Yaskawa INFORM job: R1_W63-A2(130,-90)(JEDENR)KM-OK.JBI

/JOB
//NAME R1_W63-A2(130,-90)(JEDENR)KM-OK
///FOLDERNAME KRIS-SCIANA
//POS
///NPOS 116,116,0,5,0,0
///TOOL 0
///POSTYPE PULSE
///PULSE
C00000=-63639,-75448,-57109,45781,44405,52131
C00001=-94617,-44761,-17381,50840,21971,50320
C00002=-94032,-38268,-10140,52496,20938,49575
C00003=-93501,-34314,-6346,52601,20454,49570
C00004=-93501,-33696,-5020,53682,20144,49056
C00005=-93501,-34730,-7247,51879,20668,49913
C00006=-94060,-31578,-4114,53096,20785,49286
C00007=-96769,-33900,-736,77115,20483,38452
C00008=-95613,-42258,-10455,72271,20201,40872
C00009=-114836,-25735,13136,94907,47591,35443
C00010=-113994,-25195,14177,95513,47040,35198
C00011=-113416,-25115,14231,95692,46650,35188
C00012=-114835,-25299,14106,95251,47609,35212
C00013=-114836,-25735,13136,94907,47591,35443
C00014=-120475,-35953,-1370,90254,51436,37673
C00015=-139903,-55423,-18281,79986,42519,40432
C00016=-137225,-49893,-12147,81254,40513,40051
C00017=-135734,-44853,-8428,81025,39552,40397
C00018=-135734,-43954,-6692,81758,39441,39971
C00019=-136203,-47633,-9616,81821,39746,39864
C00020=-134828,-42840,-6692,81137,38929,40458
C00021=-134687,-41796,-6081,80951,38863,40584
C00022=-135051,-44549,-7816,81347,39046,40303
C00023=-137549,-28607,9365,88397,55747,44205
C00024=-139027,-39027,1145,88234,56734,44007
C00025=-137476,-39506,859,88663,55676,44006
C00026=-139027,-39027,1145,88234,56734,44007
C00027=-137549,-29554,7549,87969,55789,44554
C00028=-148111,-23444,13104,85705,62970,44063
C00029=-149452,-24752,11123,85135,63945,44289
C00030=-152843,-27774,6403,83810,66439,44814
C00031=-190226,-72414,-43906,76175,93946,45874
C00032=-161209,-108399,-80251,28334,56751,-1893
C00033=-144499,-103217,-75669,1877,44915,-17731
C00034=-128729,-75448,-61988,-39008,44461,-40651
C00035=-127704,-59864,-42449,-54687,37585,-47688
C00036=-129098,-54028,-36168,-54912,36254,-47616
C00037=-129628,-51692,-33607,-55058,35721,-47558
C00038=-128853,-41055,-35233,-41549,49027,-56551
C00039=-128853,-40816,-34294,-41807,48684,-56370
C00040=-128840,-40622,-34262,-41768,48749,-56399
C00041=-128741,-38931,-33203,-41693,48960,-56453
C00042=-128840,-40834,-35088,-41540,49052,-56556
C00043=-127247,-51490,-28798,-68208,35092,-41834
C00044=-107460,-35727,-14488,-83818,61987,-41705
C00045=-109481,-36824,-10898,-85519,60200,-40359
C00046=-110081,-36960,-10983,-85600,59771,-40373
C00047=-108896,-36684,-10810,-85439,60617,-40344
C00048=-109015,-34543,-15794,-83164,61082,-42520
C00049=-120041,-69321,-43674,-69014,34434,-47015
C00050=-122136,-63308,-37796,-69130,32837,-47090
C00051=-122861,-57682,-33939,-68142,32556,-47661
C00052=-122861,-56927,-32189,-69156,32288,-47121
C00053=-122861,-57007,-32371,-69051,32315,-47177
C00054=-122813,-54434,-30992,-68368,32532,-47537
C00055=-123554,-57398,-33775,-67835,32116,-47869
C00056=-119901,-43791,-19123,-84492,47521,-48262
C00057=-120598,-53565,-25534,-85539,46900,-47634
C00058=-121289,-53563,-25533,-85597,46409,-47669
C00059=-119821,-53557,-25530,-85473,47449,-47596
C00060=-108619,-40866,-16292,-83893,55508,-47491
C00061=-107291,-42314,-18146,-83526,56507,-47634
C00062=-103890,-45742,-22613,-82683,59075,-47961
C00063=-65358,-57443,-36501,-72798,55432,-58639
C00064=-52417,-22993,-11744,-62287,40232,-70223
C00065=-52448,-21520,-7613,-64192,39368,-69108
C00066=-54648,-17981,-5039,-63174,38063,-69802
C00067=-53917,-7248,-3547,-52245,49316,-76029
C00068=-54705,-17968,-5209,-63027,38079,-69889
C00069=-54982,-17870,-5950,-62349,38146,-70289
C00070=-79694,-48144,-31466,-41271,33070,-83233
C00071=-77055,-57327,-41840,-41672,35586,-82928
C00072=-52399,-21595,-7667,-64214,39397,-69093
C00073=-66458,-45873,-22975,-62927,28874,-70447
C00074=-66400,-25579,1153,-60319,18878,-59217
C00075=-53020,-9869,18363,-85474,30545,-51311
C00076=-52731,-9659,19405,-86358,30690,-50818
C00077=-69612,-25105,8177,-98834,9906,-36668
C00078=-79524,-35518,1348,-134138,3863,-21977
C00079=-75482,-31811,3698,-111827,6079,-31480
C00080=-72978,-30113,4449,-103521,7442,-34705
C00081=-65283,-20283,11184,-93182,12672,-38546
C00082=-57526,-6482,21608,-89208,18094,-39567
C00083=-51529,8414,34130,-88639,22276,-39204
C00084=-53564,-8199,20742,-101222,17252,-42713
C00085=-53563,-8197,20744,-101221,17253,-42714
C00086=-52099,-17044,3865,-82598,33249,-58634
C00087=-52491,-21454,-7566,-64173,39342,-69122
C00088=-58082,-75430,-54583,-50896,47163,-49014
C00089=-107090,-97721,-77006,-13083,48945,-24888
C00090=-176270,-89310,-67424,43563,50998,31527
C00091=-192397,-7473,12373,70971,39141,64616
C00092=-198057,8223,22470,69865,43596,64795
C00093=-193600,19933,27022,52886,44499,71415
C00094=-189908,-4171,13998,69688,37731,65566
C00095=-190186,-4090,14904,70371,37727,65154
C00096=-177235,-20611,-6159,45028,35374,76862
C00097=-174898,-24503,-8833,43799,33951,77653
C00098=-192590,-382,17323,71128,53739,66386
C00099=-192440,-7538,12322,71539,53432,66088
C00100=-170167,-45771,-13804,71199,23093,66562
C00101=-167354,-31626,-8772,30750,13850,80246
C00102=-188989,-2051,16572,69929,27423,64375
C00103=-188718,-2123,15673,68886,27437,64920
C00104=-169493,-30357,-3923,58695,11001,68525
C00105=-163564,-36911,-8397,46022,7312,74716
C00106=-174644,-23722,216,62858,14603,66221
C00107=-183467,-8838,11008,67520,20712,63387
C00108=-194258,21876,37375,73130,27762,59827
C00109=-185796,4065,21904,69855,10987,63072
C00110=-187637,506,18883,71759,12230,62079
C00111=-192876,-31132,-18558,63430,41295,68875
C00112=-194286,-74397,-52359,65330,41559,67675
C00113=-215389,-105846,-76547,70055,55098,63190
C00114=-223584,-169575,-131522,59382,5921,72840
C00115=821,-169575,-131522,59382,5921,72840
BC00000=137517,4875,970976
BC00001=139957,15,947483
BC00002=139957,15,947483
BC00003=139957,15,947483
BC00004=139957,15,947483
BC00005=139957,15,947483
BC00006=139957,15,947483
BC00007=139957,15,947483
BC00008=139957,15,947483
BC00009=139957,15,947483
BC00010=139957,15,947483
BC00011=139957,15,947483
BC00012=139957,15,947483
BC00013=139957,15,947483
BC00014=139957,15,947483
BC00015=330925,15,941461
BC00016=330925,15,941461
BC00017=330925,15,941461
BC00018=330925,15,941461
BC00019=330925,15,941461
BC00020=330925,15,941461
BC00021=330925,15,941461
BC00022=330925,15,941461
BC00023=330925,15,941461
BC00024=330925,15,941461
BC00025=330925,15,941461
BC00026=330925,15,941461
BC00027=330925,15,941461
BC00028=330925,15,941461
BC00029=330925,15,941461
BC00030=330925,15,941461
BC00031=330925,15,941461
BC00032=299906,15,897004
BC00033=287499,15,879221
BC00034=269115,15,852871
BC00035=262780,15,843792
BC00036=262780,15,843792
BC00037=262780,15,843792
BC00038=262780,15,843792
BC00039=262780,15,843792
BC00040=262780,15,843792
BC00041=262780,15,843792
BC00042=262780,15,843792
BC00043=262780,15,843792
BC00044=262780,15,843792
BC00045=262780,15,843792
BC00046=262780,15,843792
BC00047=262780,15,843792
BC00048=262780,15,843792
BC00049=136654,15,835544
BC00050=136654,15,835544
BC00051=136654,15,835544
BC00052=136654,15,835544
BC00053=136654,15,835544
BC00054=136654,15,835544
BC00055=136654,15,835544
BC00056=136654,15,835544
BC00057=136654,15,835544
BC00058=136654,15,835544
BC00059=136654,15,835544
BC00060=136654,15,835544
BC00061=136654,15,835544
BC00062=136654,15,835544
BC00063=136888,15,855195
BC00064=137079,15,871196
BC00065=170526,15,870270
BC00066=169790,15,854194
BC00067=169790,15,854194
BC00068=169495,15,847764
BC00069=169495,15,847764
BC00070=169790,15,854194
BC00071=169790,15,854194
BC00072=132010,15,871427
BC00073=170892,15,872466
BC00074=110304,4966,932996
BC00075=185586,5070,932532
BC00076=185586,5070,932532
BC00077=110304,4966,932996
BC00078=149001,4966,932996
BC00079=149001,4966,932996
BC00080=185586,5070,932532
BC00081=185586,5070,932532
BC00082=185586,5070,932532
BC00083=185586,5070,932532
BC00084=195739,11327,915833
BC00085=193056,5556,931082
BC00086=200941,1554,886436
BC00087=203973,15,869264
BC00088=184133,15,878241
BC00089=216987,15,891995
BC00090=278952,15,917935
BC00091=311995,15,931768
BC00092=312647,15,915658
BC00093=312908,15,909213
BC00094=312908,15,909213
BC00095=312908,15,909213
BC00096=312908,15,909213
BC00097=312908,15,909213
BC00098=320647,15,916710
BC00099=317963,15,931959
BC00100=278547,15,932542
BC00101=318124,17,898314
BC00102=269987,15,900844
BC00103=269987,15,900844
BC00104=318124,17,898314
BC00105=268008,17,898314
BC00106=268008,17,898314
BC00107=268008,17,898314
BC00108=268008,17,898314
BC00109=259352,15,881144
BC00110=262116,15,896254
BC00111=270789,15,860195
BC00112=270789,15,860195
BC00113=270789,15,860195
BC00114=270789,15,1056585
BC00115=270789,15,1056585
///POSTYPE BASE
///RECTAN
///RCONF 0,0,0,0,1,0,0,0,0,0,0,0,0,0,0,0,0,0,0,0,0,0,0,0
P00006=2.006,1.622,-0.565,0.0000,0.0000,0.0000
P00021=0.073,2.058,-0.109,0.0000,0.0000,0.0000
P00022=2.006,1.622,-0.565,0.0000,0.0000,0.0000
///RCONF 0,0,0,0,0,0,0,0,0,0,0,0,0,0,0,0,0,0,0,0,0,0,0,0
P00023=-2.957,-4.083,2.762,0.0000,0.0000,0.0000
P00024=-1.466,-0.226,-0.419,0.0000,0.0000,0.0000
//INST
///DATE 2025/05/06 15:30
///ATTR SC,RW
///GROUP1 RB1,BS1
NOP
'r1_W63-A2(130,-90)(JEDENROBOT)
'Path S1365
SFTOF
MOVJ C00000 BC00000 VJ=20.00
MOVJ C00001 BC00001 VJ=20.00
MOVJ C00002 BC00002 VJ=20.00
MOVL C00003 BC00003 V=60.0
REFP 3 C00004 BC00004
CALL JOB:SEARCH-R1
SET P023 P006
SFTON P023
MOVL C00005 BC00005 V=60.0
REFP 3 C00006 BC00006
CALL JOB:SEARCH-R1
SET P023 P006
SFTON P023
MOVL C00007 BC00007 V=60.0
MOVL C00008 BC00008 V=60.0
MOVL C00009 BC00009 V=100.0
MOVL C00010 BC00010 V=60.0
REFP 3 C00011 BC00011
CALL JOB:SEARCH-R1
SET P023 P006
SFTON P023
MOVL C00012 BC00012 V=60.0
MOVL C00013 BC00013 V=100.0
MOVL C00014 BC00014 V=166.7
'Path S1366
SFTOF
MOVJ C00015 BC00015 VJ=20.00
MOVJ C00016 BC00016 VJ=20.00
MOVL C00017 BC00017 V=60.0
REFP 3 C00018 BC00018
CALL JOB:SEARCH-R1
SET P024 P006
SFTON P024
MOVL C00019 BC00019 V=60.0
MOVL C00020 BC00020 V=60.0
REFP 3 C00021 BC00021
CALL JOB:SEARCH-R1
SET P024 P006
SFTON P024
MOVL C00022 BC00022 V=60.0
MOVL C00023 BC00023 V=100.0
MOVL C00024 BC00024 V=60.0
REFP 3 C00025 BC00025
CALL JOB:SEARCH-R1
SET P024 P006
SFTON P024
MOVL C00026 BC00026 V=60.0
MOVL C00027 BC00027 V=100.0
MOVL C00028 BC00028 V=100.0
MOVL C00029 BC00029 V=100.0
MOVL C00030 BC00030 V=166.7
'Path VIA1504
SFTOF
MOVJ C00031 BC00031 VJ=20.00
'Path VIA1509
SFTOF
MOVJ C00032 BC00032 VJ=20.00
'Path VIA1505
SFTOF
MOVJ C00033 BC00033 VJ=20.00
'Path S1414
SFTOF
MOVJ C00034 BC00034 VJ=20.00
MOVJ C00035 BC00035 VJ=20.00
MOVJ C00036 BC00036 VJ=20.00
MOVL C00037 BC00037 V=100.0
MOVL C00038 BC00038 V=60.0
REFP 3 C00039 BC00039
CALL JOB:SEARCH-R1
SET P021 P006
SFTON P021
MOVL C00040 BC00040 V=60.0
REFP 3 C00041 BC00041
CALL JOB:SEARCH-R1
SET P021 P006
SFTON P021
MOVL C00042 BC00042 V=60.0
MOVL C00043 BC00043 V=100.0
MOVL C00044 BC00044 V=100.0
MOVL C00045 BC00045 V=60.0
REFP 3 C00046 BC00046
CALL JOB:SEARCH-R1
SET P021 P006
SFTON P021
MOVL C00047 BC00047 V=60.0
MOVL C00048 BC00048 V=100.0
'Path S1416
SFTOF
MOVJ C00049 BC00049 VJ=20.00
MOVJ C00050 BC00050 VJ=20.00
MOVL C00051 BC00051 V=60.0
REFP 3 C00052 BC00052
CALL JOB:SEARCH-R1
SET P022 P006
SFTON P022
MOVL C00053 BC00053 V=60.0
REFP 3 C00054 BC00054
CALL JOB:SEARCH-R1
SET P022 P006
SFTON P022
MOVL C00055 BC00055 V=60.0
MOVL C00056 BC00056 V=100.0
MOVL C00057 BC00057 V=60.0
REFP 3 C00058 BC00058
CALL JOB:SEARCH-R1
SET P022 P006
SFTON P022
MOVL C00059 BC00059 V=60.0
MOVL C00060 BC00060 V=100.0
MOVL C00061 BC00061 V=100.0
MOVL C00062 BC00062 V=166.7
'Path VIA1506
SFTOF
MOVJ C00063 BC00063 VJ=20.00
'Path W1380
SFTOF
SFTON P023
MOVJ C00064 BC00064 VJ=20.00
SFTOF
SFTON P023
CALL JOB:COFNIJ_DRUT
MOVJ C00065 BC00065 VJ=20.00
COMM MOVJ C00066 BC00066 VJ=20.00
COMM MOVL C00067 BC00067 V=100.0 PL=0
COMM REFP 1 C00068 BC00068
COMM REFP 2 C00069 BC00069
COMM MACRO1 MJ#(0) ARGF9
COMM ARCON
COMM MOVL C00070 BC00070 V=11.7
COMM ARCOF
COMM MOVL C00071 BC00071 V=100.0
COMM MOVL C00072 BC00072 V=166.7
COMM SFTOF
COMM 'Path W1378
COMM SFTOF
SFTOF
SFTON P023
MOVJ C00073 BC00073 VJ=20.00
MOVL C00074 BC00074 V=100.0 PL=0
REFP 1 C00075 BC00075
REFP 2 C00076 BC00076
MACRO1 MJ#(0) ARGF9
ARCON
MOVL C00077 BC00077 V=11.7
MOVL C00078 BC00078 V=11.7
MOVL C00079 BC00079 V=11.7
SFTON P024
MOVL C00080 BC00080 V=11.7
MOVL C00081 BC00081 V=11.7
MOVL C00082 BC00082 V=11.7
MOVL C00083 BC00083 V=11.7
ARCOF
MOVL C00084 BC00084 V=100.0
MOVL C00085 BC00085 V=166.7
SFTOF
'Path VIA1510
SFTOF
MOVJ C00086 BC00086 VJ=20.00
'Path W1379
SFTOF
SFTON P024
MOVJ C00087 BC00087 VJ=20.00
SFTOF
'Path VIA1507
SFTOF
MOVJ C00088 BC00088 VJ=20.00
'Path VIA1508
SFTOF
MOVJ C00089 BC00089 VJ=20.00
MOVJ C00090 BC00090 VJ=20.00
'Path W1432
SFTOF
SFTON P022
MOVJ C00091 BC00091 VJ=20.00
COMM MOVJ C00092 BC00092 VJ=20.00
COMM MOVL C00093 BC00093 V=100.0 PL=0
COMM REFP 1 C00094 BC00094
COMM REFP 2 C00095 BC00095
COMM MACRO1 MJ#(0) ARGF9
COMM ARCON
COMM MOVL C00096 BC00096 V=11.7
COMM MOVL C00097 BC00097 V=11.7
COMM ARCOF
COMM MOVL C00098 BC00098 V=100.0
COMM MOVL C00099 BC00099 V=166.7
COMM SFTOF
COMM 'Path W1433
COMM SFTOF
COMM SFTON P021
MOVJ C00100 BC00100 VJ=20.00
SFTOF
'Path W1434
SFTOF
SFTON P021
MOVL C00101 BC00101 V=100.0 PL=0
REFP 1 C00102 BC00102
REFP 2 C00103 BC00103
MACRO1 MJ#(0) ARGF9
ARCON
MOVL C00104 BC00104 V=11.7
MOVL C00105 BC00105 V=11.7
MOVL C00106 BC00106 V=11.7
SFTON P022
MOVL C00107 BC00107 V=11.7
MOVL C00108 BC00108 V=11.7
ARCOF
MOVL C00109 BC00109 V=100.0
MOVL C00110 BC00110 V=166.7
SFTOF
'Path W1435
MOVL C00111 BC00111 V=100.0
MOVL C00112 BC00112 V=166.7
SFTOF
MOVJ C00113 BC00113 VJ=20.00
MOVJ C00114 BC00114 VJ=100.00
MOVJ C00115 BC00115 VJ=100.00
END
